// TIA Portal V17 export
// export: Created 2024-09-02T12:50:04.9763277Z, ExportSetting WithDefaults, DisplayName Totally Integrated Automation Portal, DisplayVersion V17, DisplayName TIA Portal Openness, DisplayVersion V17, DisplayName TIA Portal Version Control Interface, DisplayVersion V17, DisplayName STEP 7 Professional, DisplayVersion V17, DisplayName STEP 7 Safety, DisplayVersion V17, DisplayName WinCC Professional, DisplayVersion V17
DATA_BLOCK "GraDB_SK"   // DB180
{ S7_Optimized_Access := 'TRUE'; DB_Accessible_From_OPC_UA := 'FALSE' }
AUTHOR : VAF
FAMILY : SK
NAME : SK
VERSION : 0.1
// stored: AutoNumber true, DBAccessibleFromOPCUA false, IsOnlyStoredInLoadMemory false, IsRetainMemResEnabled false, IsWriteProtectedInAS false, MemoryReserve 0
   VAR
      noAction { ExternalWritable := 'False'} : Bool;
      OP70_1 { ExternalWritable := 'False'} : Struct   // FG
         Cylinder { ExternalWritable := 'False'} : Array[1..10] of Struct   // Bereich für Gegenlüften / Area for counter ventilation
            START { ExternalWritable := 'False'} : Time;
            AKTUEL { ExternalWritable := 'False'} : Time;
         END_STRUCT;
      END_STRUCT;
      OP70_2 { ExternalWritable := 'False'} : Struct   // FG
         Cylinder { ExternalWritable := 'False'} : Array[1..10] of Struct   // Bereich für Gegenlüften / Area for counter ventilation
            START { ExternalWritable := 'False'} : Time;
            AKTUEL { ExternalWritable := 'False'} : Time;
         END_STRUCT;
      END_STRUCT;
   END_VAR
BEGIN
END_DATA_BLOCK
